// TIA Portal V19 export
FUNCTION "FC200_ServerNTP" : Void   // FC200, LAD
{ S7_Optimized_Access := 'TRUE' }
// stored: AutoNumber false, IsIECCheckEnabled true, SetENOAutomatically false
BEGIN

REGION Network 1: Server NTP (time)
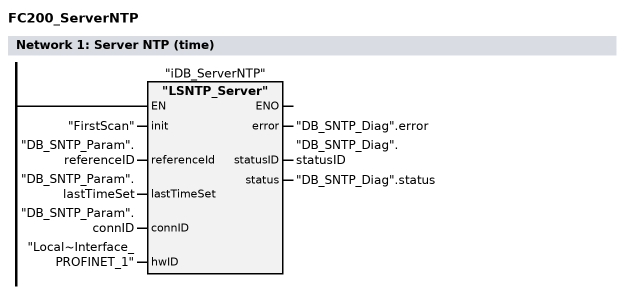
   RUNG wire#powerrail
      "iDB_ServerNTP"(init := "FirstScan", referenceId := "DB_SNTP_Param".referenceID, lastTimeSet := "DB_SNTP_Param".lastTimeSet, connID := "DB_SNTP_Param".connID, hwID := "Local~Interface_PROFINET_1", error => "DB_SNTP_Diag".error, statusID => "DB_SNTP_Diag".statusID, status => "DB_SNTP_Diag".status)
   END_RUNG
   // the same network as SCL:
   "iDB_ServerNTP"(init := "FirstScan",   // "LSNTP_Server"
                   referenceId := "DB_SNTP_Param".referenceID,
                   lastTimeSet := "DB_SNTP_Param".lastTimeSet,
                   connID := "DB_SNTP_Param".connID,
                   hwID := "Local~Interface_PROFINET_1",
                   error => "DB_SNTP_Diag".error,
                   statusID => "DB_SNTP_Diag".statusID,
                   status => "DB_SNTP_Diag".status);
END_REGION
END_FUNCTION
